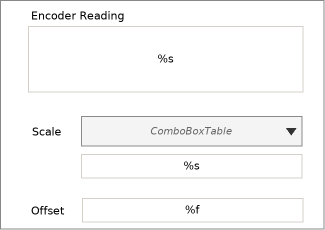
VISUALIZATION V_Encoder  // 325x230
    Textfield (28,26 275x66), "%s", text variable: Encoder.nVoltage
        p4168582468: Encoder.nVoltage
    Label (28,1 118x30), "Encoder Reading"
    Label (29,117 52x30), "Scale"
    Textfield (81,154 221x24), "%s", text variable: Encoder.nScaling
        p4168582468: Encoder.nScaling
    Label (28,196 52x30), "Offset"
    Textfield (82,198 221x24), "%f", text variable: Encoder.nOffset
        OnMouseClick: write Encoder.nOffset via VisuDialogs.Numpad, min 1, max 5000, title "Encoder Offset"
    ComboBoxTable (81,116 221x30), variable: Encoder.iScaleTable, data array: Encoder.sScalingTable
        p3854506369: Encoder.sScalingTable[INDEX]
END_VISUALIZATION

(* stored: Version 1.1.0.1, ProductVersion 3.1.4024.11
   Visu V_Encoder: Id {25ef540c-7062-415b-bb68-72c7c5628830} *)
